{attribute 'qualified_only'}
VAR_GLOBAL
	GrindingWheelMS : BOOL;
	StartGrindingWheelPB : BOOL;
	StopGrindingWheelPB : BOOL;
END_VAR

(* stored: Version 1.1.0.1, ProductVersion 3.1.4024.6
   GVL Grinder: Id {32dc2d49-9e4b-46c6-a374-c157d29889db} *)
